FUNCTION_BLOCK TGetTimeZoneInfo
VAR_INPUT
END_VAR
VAR_OUTPUT
END_VAR
VAR
    _Execution : TExecution;
    FB_GetTimeZoneInformation1 : FB_GetTimeZoneInformation;

    
END_VAR

FB_GetTimeZoneInformation1(
	sNetID:= , 
	bExecute:= _Execution.Starting, 
	tTimeout:= , 
	bBusy=> , 
	bError=> , 
	nErrID=> , 
	tzID=> , 
	tzInfo=> );
    
IF _Execution.Starting THEN
    _Execution.SetBusy();
END_IF

IF _Execution.Busy AND NOT FB_GetTimeZoneInformation1.bBusy THEN
    IF FB_GetTimeZoneInformation1.bError THEN
        _Execution.SetError(ErrorId := FB_GetTimeZoneInformation1.nErrID);
    ELSE
        _Execution.SetDone();
	END_IF
END_IF

PROPERTY Execution : IExecution
GET
Execution := _Execution;
END_GET
END_PROPERTY

PROPERTY TimeZoneInfo : ST_TimeZoneInformation
GET
TimeZoneInfo := FB_GetTimeZoneInformation1.tzInfo;
END_GET
END_PROPERTY

END_FUNCTION_BLOCK

(* stored: Version 1.1.0.1, ProductVersion 3.1.4024.3
   POU TGetTimeZoneInfo: Id {d23e141b-bc29-04fc-3517-af66238eae45}, SpecialFunc None
   Property Execution: Id {3e7e3ca9-41a5-0e3d-1cfb-58e0fc1b7aef}
   Get Get: Id {75557605-e1bf-054a-01ab-951eb37ae38e}
   Property TimeZoneInfo: Id {254f1822-6aa1-0279-1d5c-6ebe5e40f94b}
   Get Get: Id {baeed17f-0ab4-0f57-287c-e6a1b725650f} *)
